FUNCTION_BLOCK FB_STD
VAR_OUTPUT
	Out_bolRed: BOOL;
	Out_bolYellow: BOOL;
	Out_bolGreen: BOOL;
	Out_bolBlue: BOOL;
	Out_bolHorn: BOOL;
END_VAR
VAR CONSTANT
	/// Fast Toggle Blink with X ms periode
	c_BLINKFAST: UINT := 1000;
	/// Slow Toggle Blink with X ms periode
	c_BLINKSLOW: UINT := 2000;
END_VAR
VAR
	m_bolInitDone: BOOL := FALSE;
	/// Actual sample time
	m_udiSample_ms: UDINT;
	/// Actual time in ms
	m_udiTime: UDINT;
	m_bolHornEnable: BOOL := FALSE;
	m_eRed: E_LIGHTSTATE;
	m_eYellow: E_LIGHTSTATE;
	m_eGreen: E_LIGHTSTATE;
	m_eBlue: E_LIGHTSTATE;
	m_eAlarmClass: E_AlmClass;
	m_iActualState: INT;
END_VAR


IF NOT m_bolInitDone THEN
	Initialize();
END_IF

ProcessInput();
AssignTowerLights();
ProcessOutput();

{attribute 'object_name' := 'ProcessOutput'}
METHOD PROTECTED ProcessOutput : BOOL
Out_bolRed := GetOutputProcessed(m_eRed,out_bolRed);
Out_bolYellow := GetOutputProcessed(m_eYellow,out_bolYellow);
Out_bolGreen := GetOutputProcessed(m_eRed,out_bolGreen);
Out_bolBlue := GetOutputProcessed(m_eRed,out_bolBlue);
Out_bolHorn := CheckAlmClass() AND m_bolHornEnable;
END_METHOD

{attribute 'object_name' := 'ProcessInput'}
METHOD PROTECTED ProcessInput : BOOL
m_udiTime := (m_udiTime + m_udiSample_ms) MOD 1000000000;
END_METHOD

PROPERTY State : INT
SET
m_iActualState := State;
END_SET
END_PROPERTY

{attribute 'object_name' := 'GetOutputProcessed'}
METHOD PROTECTED GetOutputProcessed : BOOL
VAR_INPUT
	eColor: E_LIGHTSTATE;
	bolOutputOld: BOOL;
END_VAR
CASE eColor OF
	E_LIGHTSTATE.Off:
		GetOutputProcessed := FALSE;
	E_LIGHTSTATE.On:
		GetOutputProcessed := TRUE;
	E_LIGHTSTATE.BlinkSlow:
		IF (m_udiTime MOD c_BLINKSLOW) = 0 THEN
			GetOutputProcessed := NOT bolOutputOld;
		END_IF		
	E_LIGHTSTATE.BlinkFast:
		IF (m_udiTime MOD c_BLINKFAST) = 0 THEN
			GetOutputProcessed := NOT bolOutputOld;
		END_IF		
ELSE
	GetOutputProcessed := FALSE;
END_CASE
END_METHOD

{attribute 'object_name' := 'AssignTowerLights'}
METHOD PROTECTED AssignTowerLights : BOOL
// This method can be overwriten to get another functionality for another system.
CASE m_iActualState OF
	// RED is steady on
	// -------------------------------------------
	cSTA_DONE, 
	cSTA_INITIALIZED,
	cSTA_PONBusy,	
	cSTA_PON,		
	cSTA_EOFFBusy,	
	cSTA_EOFF,		
	cSTA_OFF:
		m_eRed 		:= E_LIGHTSTATE.On;
		m_eYellow	:= E_LIGHTSTATE.Off;
		m_eGreen	:= E_LIGHTSTATE.Off;
		m_eBlue		:= E_LIGHTSTATE.Off;		

	// Red Blink Fast	
	// -------------------------------------------
	cSTA_TSTOPBusy,	
	cSTA_TSTOP,		
	cSTA_ERROR,		
	cSTA_ERRORQuit:	
		m_eRed 		:= E_LIGHTSTATE.BlinkFast;
		m_eYellow	:= E_LIGHTSTATE.Off;
		m_eGreen	:= E_LIGHTSTATE.Off;
		m_eBlue		:= E_LIGHTSTATE.Off;		

	// Red Blink Slow	
	// -------------------------------------------
	cSTA_OFFBusy:	
		m_eRed 		:= E_LIGHTSTATE.BlinkSlow;
		m_eYellow	:= E_LIGHTSTATE.Off;
		m_eGreen	:= E_LIGHTSTATE.Off;
		m_eBlue		:= E_LIGHTSTATE.Off;		

	// Yellow Blink Slow	
	// -------------------------------------------
	cSTA_STOPBusy,	
	cSTA_INITBusy:	
		IF CheckAlmClass() THEN
			m_eRed 		:= E_LIGHTSTATE.BlinkFast;
		ELSE
			m_eRed 		:= E_LIGHTSTATE.Off;
		END_IF

		m_eYellow	:= E_LIGHTSTATE.BlinkSlow;
		m_eGreen	:= E_LIGHTSTATE.Off;
		m_eBlue		:= E_LIGHTSTATE.Off;		

	// Yellow ON	
	// -------------------------------------------
	cSTA_INIT,		
	cSTA_STOP:		
		IF CheckAlmClass() THEN
			m_eRed 		:= E_LIGHTSTATE.BlinkFast;
		ELSE
			m_eRed 		:= E_LIGHTSTATE.Off;
		END_IF

		m_eYellow	:= E_LIGHTSTATE.On;
		m_eGreen	:= E_LIGHTSTATE.Off;
		m_eBlue		:= E_LIGHTSTATE.Off;		
	
	// Green Blink Slow	
	// -------------------------------------------
	cSTA_RUNBusy:	
		IF CheckAlmClass() THEN
			m_eRed 		:= E_LIGHTSTATE.BlinkFast;
		ELSE
			m_eRed 		:= E_LIGHTSTATE.Off;
		END_IF

		m_eYellow	:= E_LIGHTSTATE.Off;
		m_eGreen	:= E_LIGHTSTATE.BlinkSlow;
		m_eBlue		:= E_LIGHTSTATE.Off;		

	// Green ON	
	// -------------------------------------------
	cSTA_RUN:		
		IF CheckAlmClass() THEN
			m_eRed 		:= E_LIGHTSTATE.BlinkFast;
		ELSE
			m_eRed 		:= E_LIGHTSTATE.Off;
		END_IF

		m_eYellow	:= E_LIGHTSTATE.Off;
		m_eGreen	:= E_LIGHTSTATE.On;
		m_eBlue		:= E_LIGHTSTATE.Off;
ELSE
	m_eRed 		:= E_LIGHTSTATE.On;
	m_eYellow	:= E_LIGHTSTATE.Off;
	m_eGreen	:= E_LIGHTSTATE.Off;
	m_eBlue		:= E_LIGHTSTATE.Off;		
END_CASE
END_METHOD

{attribute 'object_name' := 'CheckAlmClass'}
METHOD PROTECTED CheckAlmClass : BOOL
CASE m_eAlarmClass OF
	E_AlmClass.OFF,
	E_AlmClass.EOFF,
	E_AlmClass.STOP,
	E_AlmClass.TSTOP:
		CheckAlmClass := TRUE;
ELSE
	CheckAlmClass := FALSE;
END_CASE
END_METHOD

{attribute 'object_name' := 'Initialize'}
METHOD Initialize : BOOL
VAR
	udiTaskCnt: UDINT;
	fbGETCURTASKINDEX: Tc2_System.GETCURTASKINDEX;
END_VAR
//automatic read out infos about FUB
udiTaskCnt := TwinCAT_SystemInfoVarList._AppInfo.TaskCnt;
fbGETCURTASKINDEX();
udiTaskCnt := fbGETCURTASKINDEX.index;
m_udiSample_ms := TwinCAT_SystemInfoVarList._TaskInfo[UDINT_TO_DINT(udiTaskCnt)].CycleTime/10000; //[ms] X[100ns]/10000 -> [ms]
m_bolInitDone := TRUE;
END_METHOD

PROPERTY AlarmClass : E_AlmClass
SET
m_eAlarmClass := AlarmClass;
END_SET
END_PROPERTY

PROPERTY HornEnable : BOOL
SET
m_bolHornEnable := HornEnable;
END_SET
GET
HornEnable := m_bolHornEnable;
END_GET
END_PROPERTY

END_FUNCTION_BLOCK

(* stored: Version 1.1.0.1, ProductVersion 3.1.0.36
   POU FB_STD: Id {1bb648d9-9320-48ee-aa00-1104f532eccc}, SpecialFunc None
   Method ProcessOutput: Id {0f73e241-afa4-4b34-97b7-2289ab143f81}
   Method ProcessInput: Id {28cad425-68ba-46d1-b920-af193dfe7578}
   Property State: Id {476a00ed-ef74-4658-837e-0a56fd52db6b}
   Set Set: Id {f9ecf29b-fc53-4512-93d4-d08b06dc3e4b}
   Method GetOutputProcessed: Id {55800798-a2ee-47d2-bc81-7113637f1c06}
   Method AssignTowerLights: Id {59cc2aef-072b-4764-9cde-e82f43060080}
   Method CheckAlmClass: Id {c36e547f-dad2-4a37-8b7a-1e713797d340}
   Method Initialize: Id {daed0ed1-9a01-45ab-b36c-7172d3879506}
   Property AlarmClass: Id {dcbfea31-89ab-46bc-9280-e6c60e70f7ff}
   Set Set: Id {554a2e15-3880-445c-bc4c-4ca704f280b0}
   Property HornEnable: Id {ea7e9a15-73bb-4840-9fda-58e950f8a4af}
   Set Set: Id {d085baa1-b0fb-4d92-a22a-c52b963b3b5a}
   Get Get: Id {edc7907b-a708-446c-946a-ea89736993d3} *)
